// TIA Portal V20 export
TYPE "LER_typeStatusEm7"
// stored: Access Published
   STRUCT
      unloadGripComplete : Bool;
      unloadClampLockComplete : Bool;
      unloadClampCuttingComplete : Bool;
      unloadJobComplete : Bool;
      radius : LReal := 122.07;
      sepaDistances : LReal := 976.56;
   END_STRUCT;
END_TYPE
